Staubli VAL3: JointTrajPtFull.pjx

--- JointTrajPtFull.pjx ---
Parameters version=s7.3 stackSize=5000 millimeterUnit=true
Program file=convert.pgx
Program file=copyArray.pgx
Program file=decode.pgx
Program file=decodeJointData.pgx
Program file=decodeShareReal.pgx
Program file=decodeSharedInt.pgx
Program file=encode.pgx
Program file=encodeJointData.pgx
Program file=encodeShareReal.pgx
Program file=encodeSharedInt.pgx
Program file=getRow.pgx
Program file=print.pgx
Program file=printArray.pgx
Data file=JointTrajPtFull.dtx
Type name=Prefix path=Disk://Prefix/Prefix.pjx
Type name=Header path=Disk://Header/Header.pjx
Type name=Body path=Disk://JTrajPtFullBody/JTrajPtFullBody.pjx

--- JointTrajPtFull.dtx ---
public Body body
  [0]
    num accelerations[10]
      [0] = 100
      [1] = 100
    num positions[10]
      [0] = 0.178024
      [1] = 0.405265
      [2] = 0.788191
      [3] = 0.125664
      [4] = 0.444186
      [5] = -0.149575
    num robotId = 92
    num sequence
    num time = 23.78133
    num validFields = 14
    num velocities[10] = 100
public Header header
  [0]
    num nMsgType = 14
    num nCommType = 3
    num nReplyCode = 1
public Prefix prefix
  [0]
    num nLength = 148
mdesc mNomSpeed

--- convert.pgx ---
public program convert(joint& x_jJoint, mdesc& x_mMdesc)
  local num l_nRadian2Deg
begin
  // SEQUENCE
  //   END_TRAJECTORY -3
  //   STOP_TRAJECTORY -4
  if body.sequence == -4
    stopMove()
    resetMotion()
  elseIf body.sequence == -3
    x_mMdesc.blend=off
    x_mMdesc.leave=0
    x_mMdesc.reach=0
  else
    x_mMdesc.blend=Cartesian
    // mm
    x_mMdesc.leave=25
    x_mMdesc.reach=25
  endIf

  l_nRadian2Deg = 180 / 3.14159265359

  // POSITION 0x02
  if bAnd(body.validFields,2) == 2
    x_jJoint.j1=body.positions[0] * l_nRadian2Deg
    x_jJoint.j2=body.positions[1] * l_nRadian2Deg
    x_jJoint.j3=body.positions[2] * l_nRadian2Deg
    x_jJoint.j4=body.positions[3] * l_nRadian2Deg
    x_jJoint.j5=body.positions[4] * l_nRadian2Deg
    x_jJoint.j6=body.positions[5] * l_nRadian2Deg
  endIf

  // default values
  x_mMdesc.accel=100
  x_mMdesc.vel=100
  x_mMdesc.decel=100
  x_mMdesc.tvel=99999
  x_mMdesc.rvel=99999

  // VELOCITY 0x04
  if bAnd(body.validFields,4) == 4
    // percent
    x_mMdesc.vel=body.velocities[0]
  endIf

  // ACCELERATION 0x08
  if bAnd(body.validFields,8) == 8
    //percent
    x_mMdesc.accel=body.accelerations[0]
    x_mMdesc.decel=body.accelerations[1]
  endIf
end

--- copyArray.pgx ---
program copyArray(num& x_nDestArray[] (dimensions=1), num& x_nIndex (dimensions=1), num& x_nSourceArray[] (dimensions=1))
  local num i
begin
  // copies whole x_nSourceArray to the greater or equal x_nDestArray
  // starting from x_nIndex, changes the x_nIndex to point to the
  // position one after the copied elements
  for i=0 to size(x_nSourceArray)-1
    x_nDestArray[x_nIndex+i]=x_nSourceArray[i]
  endFor
  x_nIndex=x_nIndex+size(x_nSourceArray)
end

--- decode.pgx ---
public program decode(num& x_nStatus (dimensions=1), num& x_nDWordBody[] (dimensions=2))
  local num l_nBodyDWordLen
  local num i
begin
  // x_nStatus
  // -1 - unsuccessful
  // 0 - successful
  x_nStatus=-1
  l_nBodyDWordLen=34
  if size(x_nDWordBody,1)!=l_nBodyDWordLen or size(x_nDWordBody,2)!=4
    put("Size of the param is: "+toString("",size(x_nDWordBody,1)))
    putln("x"+toString("",size(x_nDWordBody,2)))
    return
  endIf
  x_nStatus=0
  call decodeSharedInt(x_nStatus,body.robotId,x_nDWordBody,0)
  call decodeSharedInt(x_nStatus,body.sequence,x_nDWordBody,1)
  call decodeSharedInt(x_nStatus,body.validFields,x_nDWordBody,2)
  call decodeShareReal(x_nStatus,body.time,x_nDWordBody,3)
  call decodeJointData(x_nStatus,body.positions,x_nDWordBody,4)
  call decodeJointData(x_nStatus,body.velocities,x_nDWordBody,14)
  call decodeJointData(x_nStatus,body.accelerations,x_nDWordBody,24)
end

--- decodeJointData.pgx ---
public program decodeJointData(num& x_nStatus (dimensions=1), num& x_nJointData[] (dimensions=1), num& x_nDWordBody[] (dimensions=2), num x_nRowIndex (dimensions=1))
  local num i
begin
  if x_nStatus<0
    return
  endIf
  x_nStatus=0
  for i=0 to size(x_nJointData)-1
    call decodeShareReal(x_nStatus,x_nJointData[i],x_nDWordBody,x_nRowIndex+i)
    if x_nStatus<0
      putln("Failed to decode joint data at index: "+toString("",x_nRowIndex+i))
      return
    endIf
  endFor
end

--- decodeSharedInt.pgx ---
public program decodeSharedInt(num& x_nStatus (dimensions=1), num& x_nValue (dimensions=1), num& x_nDWordBody[] (dimensions=2), num x_nRowIndex (dimensions=1))
  local num l_nDWordBytes[4]
begin
  if x_nStatus<0
    return
  endIf
  x_nStatus=-1
  call getRow(l_nDWordBytes,x_nDWordBody,x_nRowIndex)
  x_nStatus=fromBinary(l_nDWordBytes,4,"-4l",x_nValue)
  if x_nStatus<0
    putln("Failed to decode shared int at index "+toString("",x_nRowIndex)+" with status "+toString("",x_nStatus))
  endIf
end

--- decodeShareReal.pgx ---
public program decodeShareReal(num& x_nStatus (dimensions=1), num& x_nValue (dimensions=1), num& x_nDWordBody[] (dimensions=2), num x_nRowIndex (dimensions=1))
  local num l_nDWordBytes[4]
begin
  if x_nStatus<0
    return
  endIf
  x_nStatus=-1
  call getRow(l_nDWordBytes,x_nDWordBody,x_nRowIndex)
  x_nStatus=fromBinary(l_nDWordBytes,4,"4.0l",x_nValue)
  if x_nStatus<0
    putln("Failed to decode shared float at index "+toString("",x_nRowIndex)+" with status "+toString("",x_nStatus))
  endIf
end

--- encode.pgx ---
public program encode(num& x_nStatus (dimensions=1), num& x_nOutputBuffer[] (dimensions=1))
  local num l_nDWordBytes[4]
  local num l_nBufferPos
  local num i
begin
  if x_nStatus<0
    return
  endIf
  l_nBufferPos=0
  x_nStatus=0
  call encodeSharedInt(x_nStatus,x_nOutputBuffer,l_nBufferPos,prefix.nLength)
  call encodeSharedInt(x_nStatus,x_nOutputBuffer,l_nBufferPos,header.nMsgType)
  call encodeSharedInt(x_nStatus,x_nOutputBuffer,l_nBufferPos,header.nCommType)
  call encodeSharedInt(x_nStatus,x_nOutputBuffer,l_nBufferPos,header.nReplyCode)
  call encodeSharedInt(x_nStatus,x_nOutputBuffer,l_nBufferPos,body.robotId)
  call encodeSharedInt(x_nStatus,x_nOutputBuffer,l_nBufferPos,body.sequence)
  call encodeSharedInt(x_nStatus,x_nOutputBuffer,l_nBufferPos,body.validFields)
  call encodeShareReal(x_nStatus,x_nOutputBuffer,l_nBufferPos,body.time)
  call encodeJointData(x_nStatus,x_nOutputBuffer,l_nBufferPos,body.positions)
  call encodeJointData(x_nStatus,x_nOutputBuffer,l_nBufferPos,body.velocities)
  call encodeJointData(x_nStatus,x_nOutputBuffer,l_nBufferPos,body.accelerations)
end

--- encodeJointData.pgx ---
public program encodeJointData(num& x_nStatus (dimensions=1), num& x_nOutputBuffer[] (dimensions=1), num& x_nBufferPos (dimensions=1), num& x_nJointData[] (dimensions=1))
  local num l_nDWordBytes[4]
  local num i
begin
  if x_nStatus<0
    return
  endIf
  x_nStatus=0
  for i=0 to size(x_nJointData)-1
    call encodeShareReal(x_nStatus,x_nOutputBuffer,x_nBufferPos,x_nJointData[i])
    if x_nStatus<0
      putln("Failed to encode joint data at index: "+toString("",x_nBufferPos)+" with "+toString("",x_nJointData[i]))
      return
    endIf
  endFor
end

--- encodeSharedInt.pgx ---
public program encodeSharedInt(num& x_nStatus (dimensions=1), num& x_nOutputBuffer[] (dimensions=1), num& x_nBufferPos (dimensions=1), num x_nSharedInt (dimensions=1))
  local num l_nDWordBytes[4]
  local num i
begin
  if x_nStatus<0
    return
  endIf
  x_nStatus=-1
  x_nStatus=toBinary(x_nSharedInt,1,"-4l",l_nDWordBytes)
  if x_nStatus<0
    putln("Failed to encode shared int at index: "+toString("",x_nBufferPos))
    return
  endIf
  call copyArray(x_nOutputBuffer,x_nBufferPos,l_nDWordBytes)
end

--- encodeShareReal.pgx ---
public program encodeShareReal(num& x_nStatus (dimensions=1), num& x_nOutputBuffer[] (dimensions=1), num& x_nBufferPos (dimensions=1), num x_nSharedReal (dimensions=1))
  local num l_nDWordBytes[4]
begin
  if x_nStatus<0
    return
  endIf
  x_nStatus=-1
  x_nStatus=toBinary(x_nSharedReal,1,"4.0l",l_nDWordBytes)
  if x_nStatus<0
    putln("Failed to encode shared real at index: "+toString("",x_nBufferPos)+", status: "+toString("",x_nStatus))
    return
  endIf
  call copyArray(x_nOutputBuffer,x_nBufferPos,l_nDWordBytes)

end

--- getRow.pgx ---
program getRow(num& x_nRow[] (dimensions=1), num& x_nMatrix[] (dimensions=2), num x_nRowIndex (dimensions=1))
  local num j
begin
  for j=0 to size(x_nMatrix,2)-1
    x_nRow[j]=x_nMatrix[x_nRowIndex,j]
  endFor
end

--- print.pgx ---
public program print()
begin
  putln("robot_id: "+toString("",body.robotId))
  putln("sequence: "+toString("",body.sequence))
  putln("valid_fields: "+toString("",body.validFields))
  if bAnd(body.validFields,1)==1
    putln("time: "+toString(".3",body.time))
  endIf
  if bAnd(body.validFields,2)==2
    put("positions: ")
    call printArray("1.2",body.positions)
  endIf
  if bAnd(body.validFields,4)==4
    put("velocities: ")
    call printArray("1.2",body.velocities)
  endIf
  if bAnd(body.validFields,8)==8
    put("accelerations: ")
    call printArray("1.2",body.accelerations)
  endIf
end

--- printArray.pgx ---
program printArray(string x_sFormat (dimensions=1), num& x_nArray[] (dimensions=1))
  local num i
begin
  for i=0 to size(x_nArray)-2
    put(toString(x_sFormat,x_nArray[i]))
    put(" ")
  endFor
  putln(toString(x_sFormat,x_nArray[size(x_nArray)-1]))
end
